// TIA Portal V17 export
// export: Created 2026-04-13T11:12:53.3321362Z, ExportSetting WithDefaults, DisplayName Totally Integrated Automation Portal, DisplayVersion V17 Update 4, DisplayName TIA Portal Openness, DisplayVersion V17 Update 4, DisplayName TIA Portal Version Control Interface, DisplayVersion V17, DisplayName SINAMICS Startdrive Advanced, DisplayVersion V17, DisplayName SINAMICS Startdrive G130, G150, S120, S150, SINAMICS MV, S210, DisplayVersion V17, DisplayName SINAMICS Startdrive G110M, G120, G120C, G120D, G120P, G115D, DisplayVersion V17, DisplayName STEP 7 Professional, DisplayVersion V17 Update 4, DisplayName STEP 7 Safety, DisplayVersion V17, DisplayName WinCC Professional, DisplayVersion V17 Update 4
TagTable "INCIPCS2"
  INCIPCS2_1设定时间 : Real  (PLC tag INCIPCS2.1设定时间, HMI_连接_1, 1 s)
  INCIPCS2_2设定时间 : Real  (PLC tag INCIPCS2.2设定时间, HMI_连接_1, 1 s)
  INCIPCS2_3设定时间 : Real  (PLC tag INCIPCS2.3设定时间, HMI_连接_1, 1 s)
  INCIPCS2_4设定时间 : Real  (PLC tag INCIPCS2.4设定时间, HMI_连接_1, 1 s)
  INCIPCS2_5设定时间 : Real  (PLC tag INCIPCS2.5设定时间, HMI_连接_1, 1 s)
  INCIPCS2_6设定时间 : Real  (PLC tag INCIPCS2.6设定时间, HMI_连接_1, 1 s)
  INCIPCS2_7设定时间 : Real  (PLC tag INCIPCS2.7设定时间, HMI_连接_1, 1 s)
  INCIPCS2_8设定时间 : Real  (PLC tag INCIPCS2.8设定时间, HMI_连接_1, 1 s)
  INCIPCS2_9设定时间 : Real  (PLC tag INCIPCS2.9设定时间, HMI_连接_1, 1 s)
  INCIPCS2_10设定时间 : Real  (PLC tag INCIPCS2.10设定时间, HMI_连接_1, 1 s)
  INCIPCS2_11设定时间 : Real  (PLC tag INCIPCS2.11设定时间, HMI_连接_1, 1 s)
  INCIPCS2_12设定时间 : Real  (PLC tag INCIPCS2.12设定时间, HMI_连接_1, 1 s)
  INCIPCS2_13设定时间 : Real  (PLC tag INCIPCS2.13设定时间, HMI_连接_1, 1 s)
  INCIPCS2_14设定时间 : Real  (PLC tag INCIPCS2.14设定时间, HMI_连接_1, 1 s)
  INCIPCS2_15设定时间 : Real  (PLC tag INCIPCS2.15设定时间, HMI_连接_1, 1 s)
  INCIPCS2_16设定时间 : Real  (PLC tag INCIPCS2.16设定时间, HMI_连接_1, 1 s)
  INCIPCS2_1计时 : Real  (PLC tag INCIPCS2.1计时, HMI_连接_1, 1 s)
  INCIPCS2_2计时 : Real  (PLC tag INCIPCS2.2计时, HMI_连接_1, 1 s)
  INCIPCS2_3计时 : Real  (PLC tag INCIPCS2.3计时, HMI_连接_1, 1 s)
  INCIPCS2_4计时 : Real  (PLC tag INCIPCS2.4计时, HMI_连接_1, 1 s)
  INCIPCS2_5计时 : Real  (PLC tag INCIPCS2.5计时, HMI_连接_1, 1 s)
  INCIPCS2_6计时 : Real  (PLC tag INCIPCS2.6计时, HMI_连接_1, 1 s)
  INCIPCS2_7计时 : Real  (PLC tag INCIPCS2.7计时, HMI_连接_1, 1 s)
  INCIPCS2_8计时 : Real  (PLC tag INCIPCS2.8计时, HMI_连接_1, 1 s)
  INCIPCS2_9计时 : Real  (PLC tag INCIPCS2.9计时, HMI_连接_1, 1 s)
  INCIPCS2_10计时 : Real  (PLC tag INCIPCS2.10计时, HMI_连接_1, 1 s)
  INCIPCS2_11计时 : Real  (PLC tag INCIPCS2.11计时, HMI_连接_1, 1 s)
  INCIPCS2_12计时 : Real  (PLC tag INCIPCS2.12计时, HMI_连接_1, 1 s)
  INCIPCS2_13计时 : Real  (PLC tag INCIPCS2.13计时, HMI_连接_1, 1 s)
  INCIPCS2_14计时 : Real  (PLC tag INCIPCS2.14计时, HMI_连接_1, 1 s)
  INCIPCS2_15计时 : Real  (PLC tag INCIPCS2.15计时, HMI_连接_1, 1 s)
  INCIPCS2_16计时 : Real  (PLC tag INCIPCS2.16计时, HMI_连接_1, 1 s)
  INCIPCS2_1电导率 : Real  (PLC tag INCIPCS2.1电导率, HMI_连接_1, 1 s)
  INCIPCS2_2电导率 : Real  (PLC tag INCIPCS2.2电导率, HMI_连接_1, 1 s)
  INCIPCS2_3电导率 : Real  (PLC tag INCIPCS2.3电导率, HMI_连接_1, 1 s)
  INCIPCS2_4电导率 : Real  (PLC tag INCIPCS2.4电导率, HMI_连接_1, 1 s)
  INCIPCS2_5电导率 : Real  (PLC tag INCIPCS2.5电导率, HMI_连接_1, 1 s)
  INCIPCS2_6电导率 : Real  (PLC tag INCIPCS2.6电导率, HMI_连接_1, 1 s)
  INCIPCS2_7电导率 : Real  (PLC tag INCIPCS2.7电导率, HMI_连接_1, 1 s)
  INCIPCS2_8电导率 : Real  (PLC tag INCIPCS2.8电导率, HMI_连接_1, 1 s)
  INCIPCS2_9电导率 : Real  (PLC tag INCIPCS2.9电导率, HMI_连接_1, 1 s)
  INCIPCS2_10电导率 : Real  (PLC tag INCIPCS2.10电导率, HMI_连接_1, 1 s)
  INCIPCS2_11电导率 : Real  (PLC tag INCIPCS2.11电导率, HMI_连接_1, 1 s)
  INCIPCS2_12电导率 : Real  (PLC tag INCIPCS2.12电导率, HMI_连接_1, 1 s)
  INCIPCS2_13电导率 : Real  (PLC tag INCIPCS2.13电导率, HMI_连接_1, 1 s)
  INCIPCS2_14电导率 : Real  (PLC tag INCIPCS2.14电导率, HMI_连接_1, 1 s)
  INCIPCS2_15电导率 : Real  (PLC tag INCIPCS2.15电导率, HMI_连接_1, 1 s)
  INCIPCS2_16电导率 : Real  (PLC tag INCIPCS2.16电导率, HMI_连接_1, 1 s)
  INCIPCS2_1清洗状态 : Bool  (PLC tag INCIPCS2.1清洗状态, HMI_连接_1, 1 s)
  INCIPCS2_2清洗状态 : Bool  (PLC tag INCIPCS2.2清洗状态, HMI_连接_1, 1 s)
  INCIPCS2_3清洗状态 : Bool  (PLC tag INCIPCS2.3清洗状态, HMI_连接_1, 1 s)
  INCIPCS2_4清洗状态 : Bool  (PLC tag INCIPCS2.4清洗状态, HMI_连接_1, 1 s)
  INCIPCS2_5清洗状态 : Bool  (PLC tag INCIPCS2.5清洗状态, HMI_连接_1, 1 s)
  INCIPCS2_6清洗状态 : Bool  (PLC tag INCIPCS2.6清洗状态, HMI_连接_1, 1 s)
  INCIPCS2_7清洗状态 : Bool  (PLC tag INCIPCS2.7清洗状态, HMI_连接_1, 1 s)
  INCIPCS2_8清洗状态 : Bool  (PLC tag INCIPCS2.8清洗状态, HMI_连接_1, 1 s)
  INCIPCS2_9清洗状态 : Bool  (PLC tag INCIPCS2.9清洗状态, HMI_连接_1, 1 s)
  INCIPCS2_10清洗状态 : Bool  (PLC tag INCIPCS2.10清洗状态, HMI_连接_1, 1 s)
  INCIPCS2_11清洗状态 : Bool  (PLC tag INCIPCS2.11清洗状态, HMI_连接_1, 1 s)
  INCIPCS2_12清洗状态 : Bool  (PLC tag INCIPCS2.12清洗状态, HMI_连接_1, 1 s)
  INCIPCS2_13清洗状态 : Bool  (PLC tag INCIPCS2.13清洗状态, HMI_连接_1, 1 s)
  INCIPCS2_14清洗状态 : Bool  (PLC tag INCIPCS2.14清洗状态, HMI_连接_1, 1 s)
  INCIPCS2_15清洗状态 : Bool  (PLC tag INCIPCS2.15清洗状态, HMI_连接_1, 1 s)
  INCIPCS2_16清洗状态 : Bool  (PLC tag INCIPCS2.16清洗状态, HMI_连接_1, 1 s)
